LIN {X 0,Y 60.251,Z 550.357,A -85,B 0,C 180,E1 -29097.814,E2 -29097.814} C_VEL
LIN {X 0,Y 64.638,Z 548.045,A -85,B 0,C 180,E1 -29106.249,E2 -29106.249} C_VEL
LIN {X 0,Y 67.087,Z 546.538,A -85,B 0,C 180,E1 -29110.728,E2 -29110.728} C_VEL
LIN {X 0,Y 70.3,Z 543.681,A -85,B 0,C 180,E1 -29118.201,E2 -29118.201} C_VEL
LIN {X 0,Y 74.403,Z 540.303,A -85,B 0,C 180,E1 -29124.866,E2 -29124.866} C_VEL
LIN {X 0,Y 78.023,Z 537.872,A -85,B 0,C 180,E1 -29127.906,E2 -29127.906} C_VEL
LIN {X 0,Y 88.512,Z 530.765,A -85,B 0,C 180,E1 -29133.288,E2 -29133.288} C_VEL
LIN {X 0,Y 99.001,Z 522.327,A -85,B 0,C 180,E1 -29137.349,E2 -29137.349} C_VEL
LIN {X 0,Y 101.382,Z 520.192,A -85,B 0,C 180,E1 -29138.218,E2 -29138.218} C_VEL
LIN {X 0,Y 103.044,Z 516.707,A -85,B 0,C 180,E1 -29142.719,E2 -29142.719} C_VEL
LIN {X 0,Y 103.476,Z 515.723,A -85,B 0,C 180,E1 -29144.236,E2 -29144.236} C_VEL
LIN {X 0,Y 103.807,Z 513.909,A -85,B 0,C 180,E1 -29148.281,E2 -29148.281} C_VEL
LIN {X 0,Y 104.192,Z 512.496,A -85,B 0,C 180,E1 -29152.247,E2 -29152.247} C_VEL
LIN {X 0,Y 104.754,Z 511.378,A -85,B 0,C 180,E1 -29156.153,E2 -29156.153} C_VEL
LIN {X 0,Y 105.195,Z 510.789,A -85,B 0,C 180,E1 -29160,E2 -29160} C_VEL
LIN {X 0,Y 104.807,Z 511.46,A -85,B 0,C 180,E1 -29163.845,E2 -29163.845} C_VEL
LIN {X 0,Y 104.278,Z 512.678,A -85,B 0,C 180,E1 -29167.746,E2 -29167.746} C_VEL
LIN {X 0,Y 103.841,Z 514.27,A -85,B 0,C 180,E1 -29171.715,E2 -29171.715} C_VEL
LIN {X 0,Y 103.537,Z 515.544,A -85,B 0,C 180,E1 -29174.261,E2 -29174.261} C_VEL
LIN {X 0,Y 102.348,Z 518.18,A -85,B 0,C 180,E1 -29177.997,E2 -29177.997} C_VEL
LIN {X 0,Y 101.45,Z 520.048,A -85,B 0,C 180,E1 -29180.266,E2 -29180.266} C_VEL
LIN {X 0,Y 100.649,Z 521.333,A -85,B 0,C 180,E1 -29181.612,E2 -29181.612} C_VEL
LIN {X 0,Y 91.163,Z 529.275,A -85,B 0,C 180,E1 -29185.062,E2 -29185.062} C_VEL
LIN {X 0,Y 80.989,Z 536.525,A -85,B 0,C 180,E1 -29189.798,E2 -29189.798} C_VEL
LIN {X 0,Y 70.231,Z 543.041,A -85,B 0,C 180,E1 -29196.815,E2 -29196.815} C_VEL
LIN {X 0,Y 61.009,Z 547.92,A -85,B 0,C 180,E1 -29206.275,E2 -29206.275} C_VEL
LIN {X 0,Y 53.698,Z 551.31,A -85,B 0,C 180,E1 -29218.431,E2 -29218.431} C_VEL
LIN {X 0,Y 49.369,Z 553.315,A -85,B 0,C 180,E1 -29233.457,E2 -29233.457} C_VEL
LIN {X 0,Y 48.309,Z 553.973,A -85,B 0,C 180,E1 -29249.999,E2 -29249.999} C_VEL
LIN {X 0,Y 49.368,Z 553.285,A -85,B 0,C 180,E1 -29266.541,E2 -29266.541} C_VEL
LIN {X 0,Y 53.697,Z 551.254,A -85,B 0,C 180,E1 -29281.568,E2 -29281.568} C_VEL
LIN {X 0,Y 61.021,Z 547.835,A -85,B 0,C 180,E1 -29293.712,E2 -29293.712} C_VEL
LIN {X 0,Y 70.407,Z 542.857,A -85,B 0,C 180,E1 -29303.208,E2 -29303.208} C_VEL
LIN {X 0,Y 80.985,Z 536.372,A -85,B 0,C 180,E1 -29310.205,E2 -29310.205} C_VEL
LIN {X 0,Y 91.167,Z 529.088,A -85,B 0,C 180,E1 -29314.931,E2 -29314.931} C_VEL
LIN {X 0,Y 100.567,Z 521.179,A -85,B 0,C 180,E1 -29318.351,E2 -29318.351} C_VEL
LIN {X 0,Y 101.386,Z 519.85,A -85,B 0,C 180,E1 -29319.721,E2 -29319.721} C_VEL
LIN {X 0,Y 102.944,Z 516.459,A -85,B 0,C 180,E1 -29324.153,E2 -29324.153} C_VEL
LIN {X 0,Y 103.459,Z 515.226,A -85,B 0,C 180,E1 -29325.979,E2 -29325.979} C_VEL
LIN {X 0,Y 104.19,Z 512.467,A -85,B 0,C 180,E1 -29332.247,E2 -29332.247} C_VEL
LIN {X 0,Y 104.665,Z 511.29,A -85,B 0,C 180,E1 -29336.15,E2 -29336.15} C_VEL
LIN {X 0,Y 104.971,Z 510.685,A -85,B 0,C 180,E1 -29340,E2 -29340} C_VEL
LIN {X 0,Y 104.593,Z 511.217,A -85,B 0,C 180,E1 -29343.853,E2 -29343.853} C_VEL
LIN {X 0,Y 104.063,Z 512.303,A -85,B 0,C 180,E1 -29347.763,E2 -29347.763} C_VEL
LIN {X 0,Y 103.66,Z 513.728,A -85,B 0,C 180,E1 -29351.736,E2 -29351.736} C_VEL
LIN {X 0,Y 103.377,Z 515.509,A -85,B 0,C 180,E1 -29355.78,E2 -29355.78} C_VEL
LIN {X 0,Y 102.033,Z 518.563,A -85,B 0,C 180,E1 -29360.145,E2 -29360.145} C_VEL
LIN {X 0,Y 101.326,Z 519.962,A -85,B 0,C 180,E1 -29361.797,E2 -29361.797} C_VEL
LIN {X 0,Y 91.494,Z 528.312,A -85,B 0,C 180,E1 -29365.504,E2 -29365.504} C_VEL
LIN {X 0,Y 81.346,Z 535.568,A -85,B 0,C 180,E1 -29370.236,E2 -29370.236} C_VEL
LIN {X 0,Y 72.958,Z 540.816,A -85,B 0,C 180,E1 -29375.562,E2 -29375.562} C_VEL
LIN {X 0,Y 63.584,Z 545.902,A -85,B 0,C 180,E1 -29384.074,E2 -29384.074} C_VEL
LIN {X 0,Y 57.361,Z 548.839,A -85,B 0,C 180,E1 -29392.222,E2 -29392.222} C_VEL
LIN {X 0,Y 51.451,Z 551.526,A -85,B 0,C 180,E1 -29405.809,E2 -29405.809} C_VEL
LIN {X 0,Y 48.525,Z 552.863,A -85,B 0,C 180,E1 -29421.673,E2 -29421.673} C_VEL
LIN {X 0,Y 48.368,Z 553.035,A -85,B 0,C 180,E1 -29430.001,E2 -29430.001} C_VEL
LIN {X 0,Y 49.587,Z 552.398,A -85,B 0,C 180,E1 -29446.468,E2 -29446.468} C_VEL
LIN {X 0,Y 54.045,Z 550.426,A -85,B 0,C 180,E1 -29461.344,E2 -29461.344} C_VEL
LIN {X 0,Y 61.368,Z 547.07,A -85,B 0,C 180,E1 -29473.404,E2 -29473.404} C_VEL
LIN {X 0,Y 70.689,Z 542.231,A -85,B 0,C 180,E1 -29482.691,E2 -29482.691} C_VEL
LIN {X 0,Y 78.023,Z 537.872,A -85,B 0,C 180,E1 -29487.906,E2 -29487.906} C_VEL
LIN {X 0,Y 80.386,Z 536.201,A -85,B 0,C 180,E1 -29489.898,E2 -29489.898} C_VEL
LIN {X 0,Y 86.214,Z 530.544,A -85,B 0,C 180,E1 -29497.343,E2 -29497.343} C_VEL
LIN {X 0,Y 88.807,Z 528.47,A -85,B 0,C 180,E1 -29498.782,E2 -29498.782} C_VEL
LIN {X 0,Y 96.455,Z 522.395,A -85,B 0,C 180,E1 -29501.304,E2 -29501.304} C_VEL
LIN {X 0,Y 97.964,Z 519.775,A -85,B 0,C 180,E1 -29505.457,E2 -29505.457} C_VEL
LIN {X 0,Y 98.996,Z 516.892,A -85,B 0,C 180,E1 -29513.673,E2 -29513.673} C_VEL
LIN {X 0,Y 99.379,Z 516.305,A -85,B 0,C 180,E1 -29515.944,E2 -29515.944} C_VEL
LIN {X 0,Y 99.969,Z 515.65,A -85,B 0,C 180,E1 -29520,E2 -29520} C_VEL
LIN {X 0,Y 99.44,Z 516.385,A -85,B 0,C 180,E1 -29524.052,E2 -29524.052} C_VEL
LIN {X 0,Y 98.784,Z 517.644,A -85,B 0,C 180,E1 -29528.18,E2 -29528.18} C_VEL
LIN {X 0,Y 98.172,Z 519.314,A -85,B 0,C 180,E1 -29532.401,E2 -29532.401} C_VEL
LIN {X 0,Y 97.577,Z 520.557,A -85,B 0,C 180,E1 -29534.601,E2 -29534.601} C_VEL
LIN {X 0,Y 96.107,Z 522.966,A -85,B 0,C 180,E1 -29538.074,E2 -29538.074} C_VEL
LIN {X 0,Y 94.672,Z 524.326,A -85,B 0,C 180,E1 -29538.825,E2 -29538.825} C_VEL
LIN {X 0,Y 83.747,Z 532.522,A -85,B 0,C 180,E1 -29542.613,E2 -29542.613} C_VEL
LIN {X 0,Y 74.739,Z 538.271,A -85,B 0,C 180,E1 -29546.705,E2 -29546.705} C_VEL
LIN {X 0,Y 63.872,Z 544.194,A -85,B 0,C 180,E1 -29553.634,E2 -29553.634} C_VEL
LIN {X 0,Y 56.05,Z 547.851,A -85,B 0,C 180,E1 -29561.206,E2 -29561.206} C_VEL
LIN {X 0,Y 47.757,Z 551.241,A -85,B 0,C 180,E1 -29573.938,E2 -29573.938} C_VEL
LIN {X 0,Y 42.588,Z 553.246,A -85,B 0,C 180,E1 -29590.727,E2 -29590.727} C_VEL
LIN {X 0,Y 41.198,Z 553.904,A -85,B 0,C 180,E1 -29609.999,E2 -29609.999} C_VEL
LIN {X 0,Y 42.587,Z 553.215,A -85,B 0,C 180,E1 -29629.271,E2 -29629.271} C_VEL
LIN {X 0,Y 47.757,Z 551.184,A -85,B 0,C 180,E1 -29646.06,E2 -29646.06} C_VEL
LIN {X 0,Y 56.063,Z 547.764,A -85,B 0,C 180,E1 -29658.776,E2 -29658.776} C_VEL
LIN {X 0,Y 66.256,Z 542.851,A -85,B 0,C 180,E1 -29668.058,E2 -29668.058} C_VEL
LIN {X 0,Y 77.684,Z 536.302,A -85,B 0,C 180,E1 -29674.782,E2 -29674.782} C_VEL
LIN {X 0,Y 88.38,Z 529.017,A -85,B 0,C 180,E1 -29679.125,E2 -29679.125} C_VEL
LIN {X 0,Y 94.681,Z 524.093,A -85,B 0,C 180,E1 -29681.157,E2 -29681.157} C_VEL
LIN {X 0,Y 96.057,Z 522.73,A -85,B 0,C 180,E1 -29682.015,E2 -29682.015} C_VEL
LIN {X 0,Y 97.447,Z 520.418,A -85,B 0,C 180,E1 -29685.379,E2 -29685.379} C_VEL
LIN {X 0,Y 98.068,Z 519.141,A -85,B 0,C 180,E1 -29687.585,E2 -29687.585} C_VEL
LIN {X 0,Y 98.993,Z 516.827,A -85,B 0,C 180,E1 -29693.678,E2 -29693.678} C_VEL
LIN {X 0,Y 99.313,Z 516.22,A -85,B 0,C 180,E1 -29695.942,E2 -29695.942} C_VEL
LIN {X 0,Y 99.759,Z 515.544,A -85,B 0,C 180,E1 -29700,E2 -29700} C_VEL
LIN {X 0,Y 99.233,Z 516.147,A -85,B 0,C 180,E1 -29704.062,E2 -29704.062} C_VEL
LIN {X 0,Y 98.603,Z 517.249,A -85,B 0,C 180,E1 -29708.196,E2 -29708.196} C_VEL
LIN {X 0,Y 97.872,Z 519.565,A -85,B 0,C 180,E1 -29714.556,E2 -29714.556} C_VEL
LIN {X 0,Y 96.439,Z 522.125,A -85,B 0,C 180,E1 -29718.671,E2 -29718.671} C_VEL
LIN {X 0,Y 88.655,Z 528.383,A -85,B 0,C 180,E1 -29721.337,E2 -29721.337} C_VEL
LIN {X 0,Y 78.001,Z 535.639,A -85,B 0,C 180,E1 -29725.709,E2 -29725.709} C_VEL
LIN {X 0,Y 69.759,Z 540.48,A -85,B 0,C 180,E1 -29730.248,E2 -29730.248} C_VEL
LIN {X 0,Y 61.33,Z 544.788,A -85,B 0,C 180,E1 -29736.665,E2 -29736.665} C_VEL
LIN {X 0,Y 51.911,Z 548.908,A -85,B 0,C 180,E1 -29747.397,E2 -29747.397} C_VEL
LIN {X 0,Y 45.055,Z 551.595,A -85,B 0,C 180,E1 -29762.099,E2 -29762.099} C_VEL
LIN {X 0,Y 41.501,Z 552.932,A -85,B 0,C 180,E1 -29780.251,E2 -29780.251} C_VEL
LIN {X 0,Y 41.285,Z 553.104,A -85,B 0,C 180,E1 -29790.001,E2 -29790.001} C_VEL
LIN {X 0,Y 42.816,Z 552.467,A -85,B 0,C 180,E1 -29809.166,E2 -29809.166} C_VEL
LIN {X 0,Y 48.086,Z 550.495,A -85,B 0,C 180,E1 -29825.777,E2 -29825.777} C_VEL
LIN {X 0,Y 56.403,Z 547.138,A -85,B 0,C 180,E1 -29838.385,E2 -29838.385} C_VEL
LIN {X 0,Y 66.595,Z 542.299,A -85,B 0,C 180,E1 -29847.595,E2 -29847.595} C_VEL
LIN {X 0,Y 77.964,Z 535.822,A -85,B 0,C 180,E1 -29854.35,E2 -29854.35} C_VEL
LIN {X 0,Y 88.807,Z 528.47,A -85,B 0,C 180,E1 -29858.782,E2 -29858.782} C_VEL
LIN {X 0,Y 90.726,Z 526.826,A -85,B 0,C 180,E1 -29860.013,E2 -29860.013} C_VEL
LIN {X 0,Y 92.034,Z 525.244,A -85,B 0,C 180,E1 -29862.119,E2 -29862.119} C_VEL
LIN {X 0,Y 92.528,Z 524.271,A -85,B 0,C 180,E1 -29864.088,E2 -29864.088} C_VEL
LIN {X 0,Y 92.76,Z 523.076,A -85,B 0,C 180,E1 -29867.705,E2 -29867.705} C_VEL
LIN {X 0,Y 92.982,Z 522.122,A -85,B 0,C 180,E1 -29871.353,E2 -29871.353} C_VEL
LIN {X 0,Y 93.788,Z 520.956,A -85,B 0,C 180,E1 -29875.702,E2 -29875.702} C_VEL
LIN {X 0,Y 94.492,Z 520.274,A -85,B 0,C 180,E1 -29880,E2 -29880} C_VEL
LIN {X 0,Y 93.837,Z 521.05,A -85,B 0,C 180,E1 -29884.295,E2 -29884.295} C_VEL
LIN {X 0,Y 92.767,Z 522.837,A -85,B 0,C 180,E1 -29889.973,E2 -29889.973} C_VEL
LIN {X 0,Y 91.958,Z 524.312,A -85,B 0,C 180,E1 -29893.254,E2 -29893.254} C_VEL
LIN {X 0,Y 90.754,Z 525.678,A -85,B 0,C 180,E1 -29895.107,E2 -29895.107} C_VEL
LIN {X 0,Y 79.675,Z 533.464,A -85,B 0,C 180,E1 -29898.513,E2 -29898.513} C_VEL
LIN {X 0,Y 68.732,Z 539.863,A -85,B 0,C 180,E1 -29903.033,E2 -29903.033} C_VEL
LIN {X 0,Y 60.681,Z 543.898,A -85,B 0,C 180,E1 -29907.598,E2 -29907.598} C_VEL
LIN {X 0,Y 51.616,Z 547.782,A -85,B 0,C 180,E1 -29915.216,E2 -29915.216} C_VEL
LIN {X 0,Y 42.191,Z 551.172,A -85,B 0,C 180,E1 -29928.216,E2 -29928.216} C_VEL
LIN {X 0,Y 35.949,Z 553.177,A -85,B 0,C 180,E1 -29946.982,E2 -29946.982} C_VEL
LIN {X 0,Y 34.092,Z 553.835,A -85,B 0,C 180,E1 -29969.999,E2 -29969.999} C_VEL
LIN {X 0,Y 35.948,Z 553.146,A -85,B 0,C 180,E1 -29993.016,E2 -29993.016} C_VEL
LIN {X 0,Y 42.191,Z 551.114,A -85,B 0,C 180,E1 -30011.782,E2 -30011.782} C_VEL
LIN {X 0,Y 51.629,Z 547.694,A -85,B 0,C 180,E1 -30024.76,E2 -30024.76} C_VEL
LIN {X 0,Y 62.77,Z 542.781,A -85,B 0,C 180,E1 -30033.599,E2 -30033.599} C_VEL
LIN {X 0,Y 74.925,Z 536.231,A -85,B 0,C 180,E1 -30039.718,E2 -30039.718} C_VEL
LIN {X 0,Y 86.091,Z 528.946,A -85,B 0,C 180,E1 -30043.577,E2 -30043.577} C_VEL
LIN {X 0,Y 90.704,Z 525.508,A -85,B 0,C 180,E1 -30044.852,E2 -30044.852} C_VEL
LIN {X 0,Y 91.808,Z 524.193,A -85,B 0,C 180,E1 -30046.724,E2 -30046.724} C_VEL
LIN {X 0,Y 92.891,Z 522.221,A -85,B 0,C 180,E1 -30051.297,E2 -30051.297} C_VEL
LIN {X 0,Y 93.733,Z 520.881,A -85,B 0,C 180,E1 -30055.7,E2 -30055.7} C_VEL
LIN {X 0,Y 94.302,Z 520.164,A -85,B 0,C 180,E1 -30060,E2 -30060} C_VEL
LIN {X 0,Y 93.645,Z 520.809,A -85,B 0,C 180,E1 -30064.304,E2 -30064.304} C_VEL
LIN {X 0,Y 92.692,Z 522.277,A -85,B 0,C 180,E1 -30069.714,E2 -30069.714} C_VEL
LIN {X 0,Y 92.262,Z 523.412,A -85,B 0,C 180,E1 -30073.211,E2 -30073.211} C_VEL
LIN {X 0,Y 91.18,Z 524.826,A -85,B 0,C 180,E1 -30075.557,E2 -30075.557} C_VEL
LIN {X 0,Y 79.914,Z 532.779,A -85,B 0,C 180,E1 -30079.022,E2 -30079.022} C_VEL
LIN {X 0,Y 69.002,Z 539.183,A -85,B 0,C 180,E1 -30083.556,E2 -30083.556} C_VEL
LIN {X 0,Y 57.353,Z 544.858,A -85,B 0,C 180,E1 -30090.933,E2 -30090.933} C_VEL
LIN {X 0,Y 46.917,Z 548.978,A -85,B 0,C 180,E1 -30101.498,E2 -30101.498} C_VEL
LIN {X 0,Y 38.901,Z 551.665,A -85,B 0,C 180,E1 -30117.182,E2 -30117.182} C_VEL
LIN {X 0,Y 34.526,Z 553.001,A -85,B 0,C 180,E1 -30138.256,E2 -30138.256} C_VEL
LIN {X 0,Y 34.175,Z 553.173,A -85,B 0,C 180,E1 -30150.001,E2 -30150.001} C_VEL
LIN {X 0,Y 36.185,Z 552.535,A -85,B 0,C 180,E1 -30172.859,E2 -30172.859} C_VEL
LIN {X 0,Y 42.496,Z 550.563,A -85,B 0,C 180,E1 -30191.417,E2 -30191.417} C_VEL
LIN {X 0,Y 51.947,Z 547.207,A -85,B 0,C 180,E1 -30204.27,E2 -30204.27} C_VEL
LIN {X 0,Y 63.051,Z 542.367,A -85,B 0,C 180,E1 -30213.092,E2 -30213.092} C_VEL
LIN {X 0,Y 72.053,Z 537.694,A -85,B 0,C 180,E1 -30217.916,E2 -30217.916} C_VEL
LIN {X 0,Y 83.08,Z 530.9,A -85,B 0,C 180,E1 -30222.117,E2 -30222.117} C_VEL
LIN {X 0,Y 91.165,Z 525.063,A -85,B 0,C 180,E1 -30224.504,E2 -30224.504} C_VEL
LIN {X 0,Y 92.35,Z 523.608,A -85,B 0,C 180,E1 -30226.802,E2 -30226.802} C_VEL
LIN {X 0,Y 92.982,Z 522.122,A -85,B 0,C 180,E1 -30231.353,E2 -30231.353} C_VEL
LIN {X 0,Y 92.736,Z 521.964,A -85,B 0,C 180,E1 -30233.748,E2 -30233.748} C_VEL
LIN {X 0,Y 91.762,Z 522.491,A -85,B 0,C 180,E1 -30236.112,E2 -30236.112} C_VEL
LIN {X 0,Y 88.124,Z 525.264,A -85,B 0,C 180,E1 -30243.44,E2 -30243.44} C_VEL
LIN {X 0,Y 87.957,Z 525.456,A -85,B 0,C 180,E1 -30244.323,E2 -30244.323} C_VEL
LIN {X 0,Y 86.916,Z 526.88,A -85,B 0,C 180,E1 -30249.306,E2 -30249.306} C_VEL
LIN {X 0,Y 86.024,Z 527.913,A -85,B 0,C 180,E1 -30251.367,E2 -30251.367} C_VEL
LIN {X 0,Y 76.055,Z 534.406,A -85,B 0,C 180,E1 -30254.004,E2 -30254.004} C_VEL
LIN {X 0,Y 66.263,Z 539.795,A -85,B 0,C 180,E1 -30257.337,E2 -30257.337} C_VEL
LIN {X 0,Y 53.758,Z 545.47,A -85,B 0,C 180,E1 -30263.772,E2 -30263.772} C_VEL
LIN {X 0,Y 42.278,Z 549.587,A -85,B 0,C 180,E1 -30273.779,E2 -30273.779} C_VEL
LIN {X 0,Y 32.842,Z 552.276,A -85,B 0,C 180,E1 -30290.059,E2 -30290.059} C_VEL
LIN {X 0,Y 27.487,Z 553.604,A -85,B 0,C 180,E1 -30315.184,E2 -30315.184} C_VEL
LIN {X 0,Y 27,Z 553.766,A -85,B 0,C 180,E1 -30329.999,E2 -30329.999} C_VEL
LIN {X 0,Y 29.511,Z 553.076,A -85,B 0,C 180,E1 -30358.442,E2 -30358.442} C_VEL
LIN {X 0,Y 37.169,Z 551.044,A -85,B 0,C 180,E1 -30379.14,E2 -30379.14} C_VEL
LIN {X 0,Y 47.862,Z 547.624,A -85,B 0,C 180,E1 -30391.767,E2 -30391.767} C_VEL
LIN {X 0,Y 59.932,Z 542.71,A -85,B 0,C 180,E1 -30399.737,E2 -30399.737} C_VEL
LIN {X 0,Y 72.757,Z 536.16,A -85,B 0,C 180,E1 -30405.005,E2 -30405.005} C_VEL
LIN {X 0,Y 84.352,Z 528.875,A -85,B 0,C 180,E1 -30408.231,E2 -30408.231} C_VEL
LIN {X 0,Y 86.025,Z 527.695,A -85,B 0,C 180,E1 -30408.627,E2 -30408.627} C_VEL
LIN {X 0,Y 86.778,Z 526.757,A -85,B 0,C 180,E1 -30410.679,E2 -30410.679} C_VEL
LIN {X 0,Y 87.851,Z 525.329,A -85,B 0,C 180,E1 -30415.412,E2 -30415.412} C_VEL
LIN {X 0,Y 88.61,Z 524.53,A -85,B 0,C 180,E1 -30420,E2 -30420} C_VEL
LIN {X 0,Y 87.802,Z 525.224,A -85,B 0,C 180,E1 -30424.591,E2 -30424.591} C_VEL
LIN {X 0,Y 86.888,Z 526.398,A -85,B 0,C 180,E1 -30429.31,E2 -30429.31} C_VEL
LIN {X 0,Y 86.196,Z 527.348,A -85,B 0,C 180,E1 -30431.925,E2 -30431.925} C_VEL
LIN {X 0,Y 76.235,Z 533.854,A -85,B 0,C 180,E1 -30434.541,E2 -30434.541} C_VEL
LIN {X 0,Y 64.389,Z 540.306,A -85,B 0,C 180,E1 -30438.808,E2 -30438.808} C_VEL
LIN {X 0,Y 54.033,Z 544.928,A -85,B 0,C 180,E1 -30444.431,E2 -30444.431} C_VEL
LIN {X 0,Y 42.536,Z 549.048,A -85,B 0,C 180,E1 -30454.299,E2 -30454.299} C_VEL
LIN {X 0,Y 33.128,Z 551.734,A -85,B 0,C 180,E1 -30470.474,E2 -30470.474} C_VEL
LIN {X 0,Y 27.624,Z 553.07,A -85,B 0,C 180,E1 -30495.262,E2 -30495.262} C_VEL
LIN {X 0,Y 27.07,Z 553.242,A -85,B 0,C 180,E1 -30510.001,E2 -30510.001} C_VEL
LIN {X 0,Y 29.748,Z 552.604,A -85,B 0,C 180,E1 -30538.199,E2 -30538.199} C_VEL
LIN {X 0,Y 37.44,Z 550.632,A -85,B 0,C 180,E1 -30558.666,E2 -30558.666} C_VEL
LIN {X 0,Y 48.137,Z 547.275,A -85,B 0,C 180,E1 -30571.165,E2 -30571.165} C_VEL
LIN {X 0,Y 60.153,Z 542.436,A -85,B 0,C 180,E1 -30579.179,E2 -30579.179} C_VEL
LIN {X 0,Y 72.938,Z 535.957,A -85,B 0,C 180,E1 -30584.487,E2 -30584.487} C_VEL
LIN {X 0,Y 84.505,Z 528.741,A -85,B 0,C 180,E1 -30587.746,E2 -30587.746} C_VEL
LIN {X 0,Y 86.176,Z 527.586,A -85,B 0,C 180,E1 -30588.141,E2 -30588.141} C_VEL
LIN {X 0,Y 86.999,Z 526.557,A -85,B 0,C 180,E1 -30590.702,E2 -30590.702} C_VEL
LIN {X 0,Y 87.91,Z 525.381,A -85,B 0,C 180,E1 -30595.414,E2 -30595.414} C_VEL
LIN {X 0,Y 88.79,Z 524.634,A -85,B 0,C 180,E1 -30600,E2 -30600} C_VEL
LIN {X 0,Y 87.957,Z 525.456,A -85,B 0,C 180,E1 -30604.323,E2 -30604.323} C_VEL
LIN {X 0,Y 87.179,Z 526.158,A -85,B 0,C 180,E1 -30605.733,E2 -30605.733} C_VEL
LIN {X 0,Y 85.235,Z 527.671,A -85,B 0,C 180,E1 -30607.027,E2 -30607.027} C_VEL
LIN {X 0,Y 81.65,Z 530.125,A -85,B 0,C 180,E1 -30608.089,E2 -30608.089} C_VEL
LIN {X 0,Y 71.092,Z 536.337,A -85,B 0,C 180,E1 -30609.493,E2 -30609.493} C_VEL
LIN {X 0,Y 57.827,Z 542.769,A -85,B 0,C 180,E1 -30613.518,E2 -30613.518} C_VEL
LIN {X 0,Y 44.917,Z 547.645,A -85,B 0,C 180,E1 -30620.146,E2 -30620.146} C_VEL
LIN {X 0,Y 32.943,Z 551.035,A -85,B 0,C 180,E1 -30631.42,E2 -30631.42} C_VEL
LIN {X 0,Y 23.492,Z 553.039,A -85,B 0,C 180,E1 -30653.247,E2 -30653.247} C_VEL
LIN {X 0,Y 19.897,Z 553.697,A -85,B 0,C 180,E1 -30689.998,E2 -30689.998} C_VEL
LIN {X 0,Y 23.491,Z 553.007,A -85,B 0,C 180,E1 -30726.75,E2 -30726.75} C_VEL
LIN {X 0,Y 32.943,Z 550.974,A -85,B 0,C 180,E1 -30748.575,E2 -30748.575} C_VEL
LIN {X 0,Y 44.926,Z 547.554,A -85,B 0,C 180,E1 -30759.817,E2 -30759.817} C_VEL
LIN {X 0,Y 57.849,Z 542.64,A -85,B 0,C 180,E1 -30766.386,E2 -30766.386} C_VEL
LIN {X 0,Y 71.245,Z 536.09,A -85,B 0,C 180,E1 -30770.555,E2 -30770.555} C_VEL
LIN {X 0,Y 80.65,Z 530.463,A -85,B 0,C 180,E1 -30772.563,E2 -30772.563} C_VEL
LIN {X 0,Y 81.677,Z 529.538,A -85,B 0,C 180,E1 -30775.064,E2 -30775.064} C_VEL
LIN {X 0,Y 82.677,Z 528.641,A -85,B 0,C 180,E1 -30780,E2 -30780} C_VEL
LIN {X 0,Y 81.326,Z 529.745,A -85,B 0,C 180,E1 -30786.567,E2 -30786.567} C_VEL
LIN {X 0,Y 80.192,Z 530.615,A -85,B 0,C 180,E1 -30788.11,E2 -30788.11} C_VEL
LIN {X 0,Y 68.001,Z 537.654,A -85,B 0,C 180,E1 -30790.937,E2 -30790.937} C_VEL
LIN {X 0,Y 58.012,Z 542.365,A -85,B 0,C 180,E1 -30794.264,E2 -30794.264} C_VEL
LIN {X 0,Y 45.148,Z 547.243,A -85,B 0,C 180,E1 -30800.936,E2 -30800.936} C_VEL
LIN {X 0,Y 33.18,Z 550.634,A -85,B 0,C 180,E1 -30812.089,E2 -30812.089} C_VEL
LIN {X 0,Y 23.722,Z 552.637,A -85,B 0,C 180,E1 -30833.665,E2 -30833.665} C_VEL
LIN {X 0,Y 19.98,Z 553.31,A -85,B 0,C 180,E1 -30870.002,E2 -30870.002} C_VEL
LIN {X 0,Y 23.715,Z 552.673,A -85,B 0,C 180,E1 -30906.351,E2 -30906.351} C_VEL
LIN {X 0,Y 33.161,Z 550.701,A -85,B 0,C 180,E1 -30927.968,E2 -30927.968} C_VEL
LIN {X 0,Y 45.136,Z 547.343,A -85,B 0,C 180,E1 -30939.109,E2 -30939.109} C_VEL
LIN {X 0,Y 57.994,Z 542.504,A -85,B 0,C 180,E1 -30945.813,E2 -30945.813} C_VEL
LIN {X 0,Y 71.365,Z 536.025,A -85,B 0,C 180,E1 -30949.999,E2 -30949.999} C_VEL
LIN {X 0,Y 80.294,Z 530.754,A -85,B 0,C 180,E1 -30951.983,E2 -30951.983} C_VEL
LIN {X 0,Y 81.441,Z 529.882,A -85,B 0,C 180,E1 -30953.464,E2 -30953.464} C_VEL
LIN {X 0,Y 82.85,Z 528.739,A -85,B 0,C 180,E1 -30960,E2 -30960} C_VEL
LIN {X 0,Y 81.753,Z 529.693,A -85,B 0,C 180,E1 -30964.931,E2 -30964.931} C_VEL
LIN {X 0,Y 80.737,Z 530.607,A -85,B 0,C 180,E1 -30967.413,E2 -30967.413} C_VEL
LIN {X 0,Y 71.092,Z 536.337,A -85,B 0,C 180,E1 -30969.493,E2 -30969.493} C_VEL
LIN {X 0,Y 65.879,Z 538.998,A -85,B 0,C 180,E1 -30970.267,E2 -30970.267} C_VEL
LIN {X 0,Y 56.776,Z 542.894,A -85,B 0,C 180,E1 -30970.198,E2 -30970.198} C_VEL
LIN {X 0,Y 47.451,Z 546.213,A -85,B 0,C 180,E1 -30970.198,E2 -30970.198} C_VEL
LIN {X 0,Y 41.91,Z 547.877,A -85,B 0,C 180,E1 -30971.667,E2 -30971.667} C_VEL
LIN {X 0,Y 29.852,Z 550.966,A -85,B 0,C 180,E1 -30979.652,E2 -30979.652} C_VEL
LIN {X 0,Y 18.291,Z 552.971,A -85,B 0,C 180,E1 -30999.781,E2 -30999.781} C_VEL
LIN {X 0,Y 12.786,Z 553.628,A -85,B 0,C 180,E1 -31049.997,E2 -31049.997} C_VEL
LIN {X 0,Y 18.29,Z 552.938,A -85,B 0,C 180,E1 -31100.216,E2 -31100.216} C_VEL
LIN {X 0,Y 29.851,Z 550.905,A -85,B 0,C 180,E1 -31120.342,E2 -31120.342} C_VEL
LIN {X 0,Y 42.989,Z 547.484,A -85,B 0,C 180,E1 -31128.78,E2 -31128.78} C_VEL
LIN {X 0,Y 56.594,Z 542.569,A -85,B 0,C 180,E1 -31133.442,E2 -31133.442} C_VEL
LIN {X 0,Y 66.953,Z 537.832,A -85,B 0,C 180,E1 -31135.709,E2 -31135.709} C_VEL
LIN {X 0,Y 74.948,Z 533.483,A -85,B 0,C 180,E1 -31136.953,E2 -31136.953} C_VEL
LIN {X 0,Y 76.139,Z 532.737,A -85,B 0,C 180,E1 -31138.44,E2 -31138.44} C_VEL
LIN {X 0,Y 76.528,Z 532.477,A -85,B 0,C 180,E1 -31140,E2 -31140} C_VEL
LIN {X 0,Y 76.098,Z 532.722,A -85,B 0,C 180,E1 -31141.864,E2 -31141.864} C_VEL
LIN {X 0,Y 74.927,Z 533.435,A -85,B 0,C 180,E1 -31143.66,E2 -31143.66} C_VEL
LIN {X 0,Y 63.553,Z 539.394,A -85,B 0,C 180,E1 -31145.579,E2 -31145.579} C_VEL
LIN {X 0,Y 49.857,Z 545.068,A -85,B 0,C 180,E1 -31149.343,E2 -31149.343} C_VEL
LIN {X 0,Y 36.467,Z 549.187,A -85,B 0,C 180,E1 -31155.507,E2 -31155.507} C_VEL
LIN {X 0,Y 23.916,Z 551.874,A -85,B 0,C 180,E1 -31168.17,E2 -31168.17} C_VEL
LIN {X 0,Y 14.349,Z 553.208,A -85,B 0,C 180,E1 -31200.677,E2 -31200.677} C_VEL
LIN {X 0,Y 12.878,Z 553.379,A -85,B 0,C 180,E1 -31230.003,E2 -31230.003} C_VEL
LIN {X 0,Y 18.477,Z 552.742,A -85,B 0,C 180,E1 -31279.533,E2 -31279.533} C_VEL
LIN {X 0,Y 29.993,Z 550.769,A -85,B 0,C 180,E1 -31299.605,E2 -31299.605} C_VEL
LIN {X 0,Y 43.109,Z 547.411,A -85,B 0,C 180,E1 -31308.015,E2 -31308.015} C_VEL
LIN {X 0,Y 56.821,Z 542.508,A -85,B 0,C 180,E1 -31312.894,E2 -31312.894} C_VEL
LIN {X 0,Y 70.478,Z 536.092,A -85,B 0,C 180,E1 -31315.715,E2 -31315.715} C_VEL
LIN {X 0,Y 75.061,Z 533.546,A -85,B 0,C 180,E1 -31316.41,E2 -31316.41} C_VEL
LIN {X 0,Y 76.223,Z 532.839,A -85,B 0,C 180,E1 -31318.161,E2 -31318.161} C_VEL
LIN {X 0,Y 76.665,Z 532.586,A -85,B 0,C 180,E1 -31320,E2 -31320} C_VEL
LIN {X 0,Y 76.262,Z 532.853,A -85,B 0,C 180,E1 -31321.566,E2 -31321.566} C_VEL
LIN {X 0,Y 73.591,Z 534.456,A -85,B 0,C 180,E1 -31323.248,E2 -31323.248} C_VEL
LIN {X 0,Y 60.033,Z 541.267,A -85,B 0,C 180,E1 -31325.675,E2 -31325.675} C_VEL
LIN {X 0,Y 46.357,Z 546.509,A -85,B 0,C 180,E1 -31329.786,E2 -31329.786} C_VEL
LIN {X 0,Y 41.91,Z 547.877,A -85,B 0,C 180,E1 -31331.667,E2 -31331.667} C_VEL
LIN {X 0,Y 36.333,Z 549.402,A -85,B 0,C 180,E1 -31333.595,E2 -31333.595} C_VEL
LIN {X 0,Y 26.636,Z 551.353,A -85,B 0,C 180,E1 -31334.845,E2 -31334.845} C_VEL
LIN {X 0,Y 18.779,Z 552.457,A -85,B 0,C 180,E1 -31336.287,E2 -31336.287} C_VEL
LIN {X 0,Y 13.072,Z 553.049,A -85,B 0,C 180,E1 -31341.702,E2 -31341.702} C_VEL
LIN {X 0,Y 11.315,Z 553.175,A -85,B 0,C 180,E1 -31345.894,E2 -31345.894} C_VEL
LIN {X 0,Y 5.688,Z 553.559,A -85,B 0,C 180,E1 -31409.993,E2 -31409.993} C_VEL
LIN {X 0,Y 14.781,Z 552.868,A -85,B 0,C 180,E1 -31481.975,E2 -31481.975} C_VEL
LIN {X 0,Y 28.262,Z 550.835,A -85,B 0,C 180,E1 -31494.08,E2 -31494.08} C_VEL
LIN {X 0,Y 42.185,Z 547.414,A -85,B 0,C 180,E1 -31498.327,E2 -31498.327} C_VEL
LIN {X 0,Y 50.898,Z 544.546,A -85,B 0,C 180,E1 -31500.001,E2 -31500.001} C_VEL
LIN {X 0,Y 49.205,Z 545.138,A -85,B 0,C 180,E1 -31501.132,E2 -31501.132} C_VEL
LIN {X 0,Y 35.239,Z 549.257,A -85,B 0,C 180,E1 -31504.301,E2 -31504.301} C_VEL
LIN {X 0,Y 21.492,Z 551.943,A -85,B 0,C 180,E1 -31511.189,E2 -31511.189} C_VEL
LIN {X 0,Y 8.861,Z 553.277,A -85,B 0,C 180,E1 -31537.531,E2 -31537.531} C_VEL
LIN {X 0,Y 5.77,Z 553.448,A -85,B 0,C 180,E1 -31590.007,E2 -31590.007} C_VEL
LIN {X 0,Y 14.873,Z 552.81,A -85,B 0,C 180,E1 -31660.929,E2 -31660.929} C_VEL
LIN {X 0,Y 28.308,Z 550.838,A -85,B 0,C 180,E1 -31673.267,E2 -31673.267} C_VEL
LIN {X 0,Y 42.207,Z 547.48,A -85,B 0,C 180,E1 -31677.561,E2 -31677.561} C_VEL
LIN {X 0,Y 49.206,Z 545.254,A -85,B 0,C 180,E1 -31678.915,E2 -31678.915} C_VEL
LIN {X 0,Y 50.043,Z 544.964,A -85,B 0,C 180,E1 -31679.999,E2 -31679.999} C_VEL
LIN {X 0,Y 40.199,Z 548.041,A -85,B 0,C 180,E1 -31682.071,E2 -31682.071} C_VEL
LIN {X 0,Y 28.263,Z 550.898,A -85,B 0,C 180,E1 -31685.912,E2 -31685.912} C_VEL
LIN {X 0,Y 14.782,Z 552.902,A -85,B 0,C 180,E1 -31698.023,E2 -31698.023} C_VEL
LIN {X 0,Y 11.315,Z 553.175,A -85,B 0,C 180,E1 -31705.894,E2 -31705.894} C_VEL
LIN {X 0,Y 9.774,Z 555.17,A -85,B 0,C 180,E1 -31711.57,E2 -31711.57} C_VEL
LIN {X 0,Y 9.774,Z 600,A -85,B 0,C 180,E1 -31711.57,E2 -31711.57} C_VEL
LIN {X 0,Y 9.774,Z 600,A -85,B 0,C 180,E1 -31711.57,E2 -31711.57}

QRS_NEXT_CUT()

QRS_NEXT()
QRS_HOME()

END
